FUNCTION_BLOCK Xenon1900VirtualCom
VAR
	_bConnect				:BOOL;
	_ComCfg					:ComSerialConfig;
	_TxBuffer				:ComBuffer;
	_RxBuffer				:ComBuffer;
	_SerialLineControlADS	:SerialLineControlADS;
	_bReset					:BOOL;
	_sStringData			:STRING;
	_ReceiveString			:ReceiveString;

END_VAR

_SerialLineControlADS(
	Connect		:= _bConnect, 
	SerialCfg	:= _ComCfg, 
	NetId		:= '', 
	Timeout		:= DEFAULT_ADS_TIMEOUT, 
	TxBuffer	:= _TxBuffer, 
	RxBuffer	:= _RxBuffer);

_ReceiveString(
	Prefix			:= '', 
	Suffix			:= '', 
	Timeout			:= T#250ms, 
	Reset			:= _bReset, 
	ReceivedString	:= _sStringData, 
	RXbuffer		:= _RxBuffer);

PROPERTY PUBLIC bConnect : BOOL
SET
_bConnect := bConnect;
END_SET
END_PROPERTY

PROPERTY PUBLIC bStringReceived : BOOL
GET
VAR_OUTPUT
END_VAR
VAR
END_VAR
bStringReceived := _ReceiveString.StringReceived;
END_GET
END_PROPERTY

PROPERTY PUBLIC sStringData : STRING
GET
sStringData := _sStringData;
END_GET
END_PROPERTY

PROPERTY PUBLIC uiComPort : UINT
SET
_ComCfg.ComPort := UINT_TO_UDINT(uiComPort);
END_SET
END_PROPERTY

END_FUNCTION_BLOCK

(* stored: Version 1.1.0.1
   POU Xenon1900VirtualCom: Id {df0a461f-910b-4b9a-ad19-6b03e7d3cca0}, SpecialFunc None
   Folder Properties: Id {77a37cba-d5f3-4393-ab36-3994d78c56dc}
   Property bConnect: Id {4a4aa5f5-8518-4233-8b33-7499164edd53}
   Set Set: Id {f6004e24-8893-4487-ab35-47477e2a46fd}
   Property bStringReceived: Id {68d72b70-9f8a-4928-a1b1-be0257d73ca7}
   Get Get: Id {444dcc77-88e5-4707-895d-bd54a6b8664a}
   Property sStringData: Id {bc370157-2d55-4c9d-bad8-11359222fdb2}
   Get Get: Id {4b93631f-cc5f-4cd5-9d46-15c383957d94}
   Property uiComPort: Id {a0fab9b3-04d8-43dd-ab0a-c7a43451de24}
   Set Set: Id {a48dcd18-7756-4036-bd54-80dd2ff1c193} *)
